ABB RAPID module: 002165AD

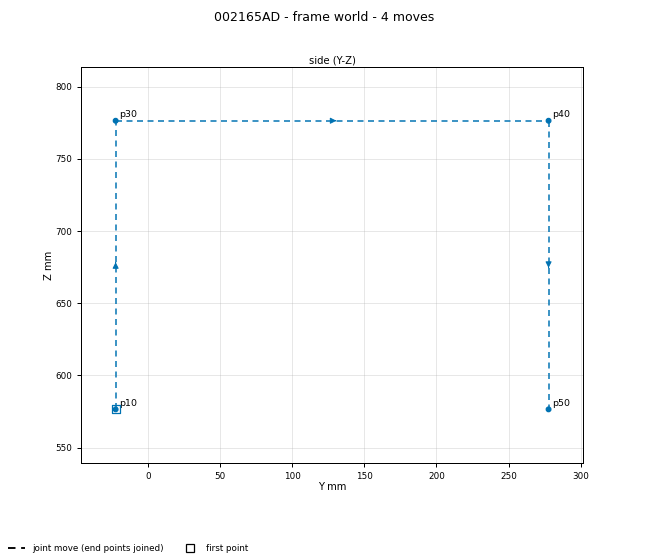
[picture p0: tool path of 002165AD in frame world, 4 of 6 moves have a stored position in this frame; points joined in program order, loops and branches not executed]
MODULE MainModule
	CONST robtarget p10:=[[924.16,-22.34,576.5],[0.0370625,-0.674596,0.737188,0.00996895],[-1,2,-4,1],[9E+09,9E+09,9E+09,9E+09,9E+09,9E+09]];
	CONST robtarget p20:=[[924.16,-22.34,576.50],[0.0370625,-0.674596,0.737188,0.00996895],[-1,2,-4,1],[9E+9,9E+9,9E+9,9E+9,9E+9,9E+9]];
	CONST robtarget p30:=[[924.16,-22.34,776.5],[0.0370629,-0.674596,0.737189,0.00996926],[-1,2,-3,1],[9E+09,9E+09,9E+09,9E+09,9E+09,9E+09]];
	CONST robtarget p40:=[[924.16,277.66,776.5],[0.0370627,-0.674596,0.737188,0.00996888],[0,2,-3,1],[9E+09,9E+09,9E+09,9E+09,9E+09,9E+09]];
	CONST robtarget p50:=[[924.16,277.66,576.5],[0.0370625,-0.674597,0.737188,0.00996883],[0,2,-3,1],[9E+09,9E+09,9E+09,9E+09,9E+09,9E+09]];
	PROC main()


		Reset do0;
		MoveAbsJ [[-5.5198,-2.10431,5.70604,183.939,-84.4136,-270.758],[9E+09,9E+09,9E+09,9E+09,9E+09,9E+09]]\NoEOffs, v1000, fine, tool0;
		MoveJ p10, v1000, fine, tool0;
		Set do0;
		MoveJ p30, v1000, fine, tool0;
		MoveJ p40, v1000, fine, tool0;
		MoveJ p50, v1000, fine, tool0;
		Reset do0;
		MoveAbsJ [[-5.5198,-2.10431,5.70604,183.939,-84.4136,-270.758],[9E+09,9E+09,9E+09,9E+09,9E+09,9E+09]]\NoEOffs, v1000, fine, tool0;
	ENDPROC
ENDMODULE
